TYPE ST_HW_STATUS_ROT :
STRUCT
	bError:BOOL:=FALSE;
	nErrorId:UDINT:=0;
	bEnabled:BOOL:=FALSE;
	eTargetState: TARGET_STATE_MACHINE;
    sErrorStr:STRING:='NO ERROR';
	fActTorque:LREAL:=0;
	fActPos:LREAL:=0;
	fActVel:LREAL:=0;	
	fActTemp:LREAL:=0;
	fSetVelRaw:LREAL;
	fBrakeActTemp1:LREAL;
	fBrakeActTemp2:LREAL;
	fPhaseOffsetActDeg:LREAL;
	bBrake1TempAlarm:BOOL;
	bBrake2TempAlarm:BOOL;
	bEStopOK:BOOL;                       // s2: ch1: emergency stop ok                 Verify: OK   
	bMainDriveThermalFilterOK:BOOL; // s2: ch2: rf01 termal braking filter OK..   Verify: Q to Markus: Maybe this should be rf02?
	bFuseMainRotationOK:BOOL;       // s2: ch6: fc01 fuse target wheel motor OK
	fRotTemp:LREAL;                 // s13: ch4: kf12 Target Main motor Temperature (KTY) (in deg*10)
	bSumILOK:BOOL:=FALSE;
	bHwStatusOK:BOOL:=FALSE;
	bManualInterlockOverride:BOOL:=FALSE;
	bGeneralILOK:BOOL:=FALSE;  // All on direction related summary interlocks
END_STRUCT
END_TYPE

(* stored: Version 1.1.0.1, ProductVersion 3.1.4024.6
   DUT ST_HW_STATUS_ROT: Id {f2d0bd80-c5ac-47d7-ab04-436fe827dce5} *)
